PROGRAM MAIN
VAR
	bRun_Process : BOOL;
	bStop_process : BOOL;
	bProcess_Status : BOOL;
	tProcess_Duration : TIME;
	fbProcess_Timer : TON;
	bTimer_Done : BOOL;	
END_VAR

//bProcess_Status := bRun_Process;

fbProcess_Timer(IN:= bProcess_Status, PT:= tProcess_Duration, Q=> bTimer_Done, ET=> );


IF bRun_Process THEN
	bProcess_Status := TRUE;
END_IF

IF bStop_Process OR bTimer_Done THEN
	bProcess_Status := FALSE;
END_IF

END_PROGRAM

(* stored: Version 1.1.0.1, ProductVersion 3.1.4024.13
   POU MAIN: Id {f71e8fc5-8849-408d-ba5b-2c650398fb9f}, SpecialFunc None *)
